// TIA Portal V19 export
FUNCTION_BLOCK "Air_Flow"   // FB131, LAD
// stored: MemoryReserve 100, SetENOAutomatically false
   VAR
      AirCounter : Real;
      Aux1s : Bool;
   END_VAR
   VAR_TEMP
      scaleRetVal : Word;
      Value : Real;
   END_VAR
BEGIN

REGION Network 1 (SCL): Air Flow / Aria compressa
   // Air Flow
   #scaleRetVal := SCALE(IN := "CC1_Ai_GeneralPressure_Air", HI_LIM := 2000.0, LO_LIM := 0.0, BIPOLAR := FALSE, OUT => #Value);
   IF (#scaleRetVal = 0)
       AND (#Value > 0.0)
   THEN
       "Air_Data".Air.Flow := #Value;
   ELSE
       "Air_Data".Air.Flow := 0.0;
   END_IF;
END_REGION

REGION Network 2 (SCL): Air Flow counter / Conteggio aria compressa
   // Flow
   #AirCounter += ("Air_Data".Air.Flow / 60000000.0) * "Sys".PreviousCycleTime; // [kNl]
END_REGION

REGION Network 3 (SCL): Consumption / Consumi
   IF TRUE
       AND "Sys".Clock_1S
       AND NOT #Aux1s
   THEN
       #Aux1s := TRUE;

       // Air Consumption
       "Air_Data".Air.TotalConsumption += #AirCounter;
       #AirCounter := 0.0;


   ELSIF TRUE
       AND NOT "Sys".Clock_1S
   THEN
       #Aux1s := FALSE;

   END_IF;
END_REGION
END_FUNCTION_BLOCK
